{attribute 'qualified_only'}
VAR_GLOBAL
	iwPumpSpeed   		AT%I* :  WORD; 	// Speed of the flow into the tank 0 - 100%
										// 40% slowly drain 50% stand still 60% filling
										

	isStatusText 		AT%I* : STRING := 'Test text'; // Text on the info display
	
	qwActualLevel 		AT%Q* : WORD;  	// Level in the tank	
	
END_VAR

(* stored: Version 1.1.0.1
   GVL GVL: Id {9198b5c0-b7ca-4c3a-96d3-3e2544de245c} *)
